Yaskawa INFORM job: clamp_07_08_23_cylinder_program.JBI

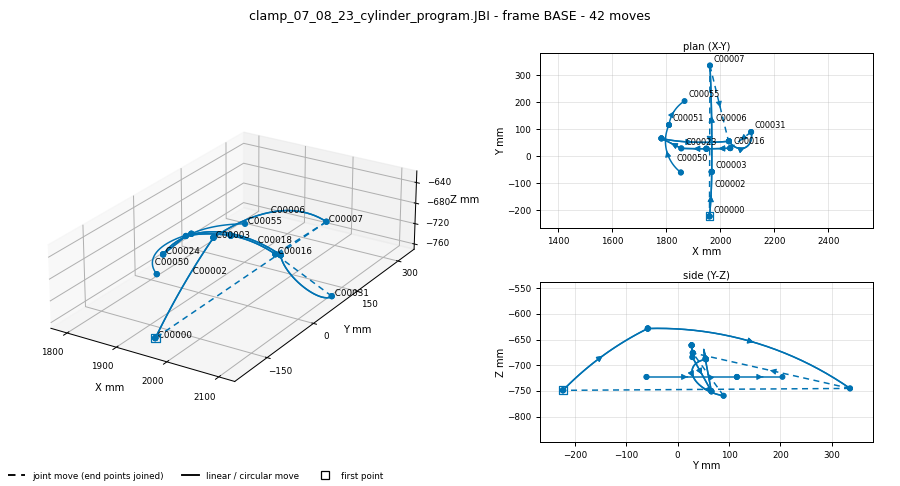
[picture p0: tool path of clamp_07_08_23_cylinder_program.JBI in frame BASE, 42 of 62 moves have a stored position in this frame; points joined in program order, loops and branches not executed]
/JOB
//NAME clamp_07_08_23_cylinder_program
//POS
///NPOS 56,0,56,0,0,0
///TOOL 0
///POSTYPE BASE
///RECTAN
///RCONF 0,0,0,0,0,0,0,0,0,0,0,0,0,0,0,0,0,0,0,0,0,0,0,0
C00000=1960.075828,-223.019615,-748.824454,180.000000,-60.000000,90.001386
C00001=1960.075828,-223.019615,-748.824454,180.000000,-60.000000,90.001386
C00002=1966.557197,-127.835510,-669.176522,-175.000000,-39.379629,92.626092
C00003=1968.376913,-58.034649,-628.612835,-161.404282,5.000000,5.000000
C00004=1968.376913,-58.034649,-628.612835,-161.404282,5.000000,5.000000
C00005=1968.376913,-58.034649,-628.612835,-161.404282,5.000000,5.000000
C00006=1968.142396,117.168535,-647.002737,151.969726,5.000000,-5.000000
C00007=1961.735097,335.262586,-745.090179,180.000000,-60.000000,-90.296572
C00008=1960.075828,-223.019615,-748.824454,180.000000,-60.000000,90.001386
C00009=1960.075828,-223.019615,-748.824454,180.000000,-60.000000,90.001386
C00010=1966.557197,-127.835510,-669.176522,-175.000000,-39.379629,92.626092
C00011=1968.376913,-58.034649,-628.612835,-161.404282,5.000000,5.000000
C00012=1968.376913,-58.034649,-628.612835,-161.404282,5.000000,5.000000
C00013=1968.376913,-58.034649,-628.612835,-161.404282,5.000000,5.000000
C00014=1968.142396,117.168535,-647.002737,151.969726,5.000000,-5.000000
C00015=1961.735097,335.262586,-745.090179,180.000000,-60.000000,-90.296572
C00016=2036.786677,29.436047,-676.031527,-174.048611,23.855296,5.000000
C00017=2036.786677,29.436047,-676.031527,-174.048611,23.855296,5.000000
C00018=1997.954834,27.911156,-664.054338,-174.328079,11.246992,5.000000
C00019=1948.764188,27.199700,-661.190386,-174.288511,-5.000000,-5.000000
C00020=1948.764188,27.199700,-661.190386,-174.288511,-5.000000,-5.000000
C00021=1948.764188,27.199700,-661.190386,-174.288511,-5.000000,-5.000000
C00022=1902.713206,27.551328,-668.774485,-173.853319,-18.487941,-5.000000
C00023=1855.573167,28.672798,-684.219428,175.000000,-33.996707,8.950518
C00024=1782.149442,65.644826,-750.764678,-180.000000,-60.000000,1.268123
C00025=1782.149442,65.644826,-750.764678,-180.000000,-60.000000,1.268123
C00026=1867.617170,53.257139,-684.581782,175.000000,-31.333075,9.869447
C00027=2031.930642,55.063888,-688.401258,-174.027335,24.456893,5.000000
C00028=2031.930642,55.063888,-688.401258,-174.027335,24.456893,5.000000
C00029=2031.930642,55.063888,-688.401258,-174.027335,24.456893,5.000000
C00030=2114.529672,61.982565,-750.948407,-175.000000,-59.425940,175.000000
C00031=2114.214530,89.330125,-759.380789,180.000000,-60.000000,-172.637609
C00032=2036.786677,29.436047,-676.031527,-174.048611,23.855296,5.000000
C00033=2036.786677,29.436047,-676.031527,-174.048611,23.855296,5.000000
C00034=1997.954834,27.911156,-664.054338,-174.328079,11.246992,5.000000
C00035=1948.764188,27.199700,-661.190386,-174.288511,-5.000000,-5.000000
C00036=1948.764188,27.199700,-661.190386,-174.288511,-5.000000,-5.000000
C00037=1948.764188,27.199700,-661.190386,-174.288511,-5.000000,-5.000000
C00038=1902.713206,27.551328,-668.774485,-173.853319,-18.487941,-5.000000
C00039=1855.573167,28.672798,-684.219428,175.000000,-33.996707,8.950518
C00040=1782.149442,65.644826,-750.764678,-180.000000,-60.000000,1.268123
C00041=1782.149442,65.644826,-750.764678,-180.000000,-60.000000,1.268123
C00042=1867.617170,53.257139,-684.581782,175.000000,-31.333075,9.869447
C00043=2031.930642,55.063888,-688.401258,-174.027335,24.456893,5.000000
C00044=2031.930642,55.063888,-688.401258,-174.027335,24.456893,5.000000
C00045=2031.930642,55.063888,-688.401258,-174.027335,24.456893,5.000000
C00046=2114.529672,61.982565,-750.948407,-175.000000,-59.425940,175.000000
C00047=2114.214530,89.330125,-759.380789,180.000000,-60.000000,-172.637609
C00048=1854.100788,-60.572273,-722.697460,180.000000,-60.000000,39.056159
C00049=1854.100788,-60.572273,-722.697460,180.000000,-60.000000,39.056159
C00050=1825.406210,-31.437250,-722.697460,180.000000,-60.000000,27.527976
C00051=1810.062104,115.232922,-722.697460,180.000000,-60.000000,-15.007935
C00052=1810.062104,115.232922,-722.697460,180.000000,-60.000000,-15.007935
C00053=1810.062104,115.232922,-722.697460,180.000000,-60.000000,-15.007935
C00054=1835.839436,175.302882,-722.697460,-180.000000,-60.000000,-33.491908
C00055=1867.753817,203.827510,-722.697460,180.000000,-60.000000,-45.587231
///POSTYPE PULSE
///PULSE
EX00000=0
EX00001=92160
EX00002=184320
EX00003=276480
///POSTYPE PULSE
///PULSE
EC00000=0
EC00001=0
EC00002=0
EC00003=0
EC00004=0
EC00005=0
EC00006=0
EC00007=0
EC00008=0
EC00009=0
EC00010=0
EC00011=0
EC00012=0
EC00013=0
EC00014=0
EC00015=0
EC00016=0
EC00017=0
EC00018=0
EC00019=0
EC00020=0
EC00021=0
EC00022=0
EC00023=0
EC00024=0
EC00025=0
EC00026=0
EC00027=0
EC00028=0
EC00029=0
EC00030=0
EC00031=0
EC00032=0
EC00033=0
EC00034=0
EC00035=0
EC00036=0
EC00037=0
EC00038=0
EC00039=0
EC00040=0
EC00041=0
EC00042=0
EC00043=0
EC00044=0
EC00045=0
EC00046=0
EC00047=0
EC00048=276480
EC00049=276480
EC00050=276480
EC00051=276480
EC00052=276480
EC00053=276480
EC00054=276480
EC00055=276480
//INST
///DATE 2023/08/07 12:02
///ATTR SC,RW,RJ
////FRAME BASE
///GROUP1 RB1,ST1
NOP
MOVJ P009 EX000 VJ=15.00
MOVJ C00000 EC00000 VJ=15.0
CALL JOB:SPYON
MOVC C00001 EC00001 V=150.0
MOVC C00002 EC00002 V=150.0
MOVC C00003 EC00003 V=150.0
MOVL C00004 EC00004 V=150.0
MOVC C00005 EC00005 V=150.0
MOVC C00006 EC00006 V=150.0
MOVC C00007 EC00007 V=150.0
CALL JOB:SPYOF
MOVJ C00008 EC00008 VJ=15.0
CALL JOB:SPYON
MOVC C00009 EC00009 V=150.0
MOVC C00010 EC00010 V=150.0
MOVC C00011 EC00011 V=150.0
MOVL C00012 EC00012 V=150.0
MOVC C00013 EC00013 V=150.0
MOVC C00014 EC00014 V=150.0
MOVC C00015 EC00015 V=150.0
CALL JOB:SPYOF
MOVJ C00016 EC00016 VJ=15.0
CALL JOB:SPYON
MOVC C00017 EC00017 V=150.0
MOVC C00018 EC00018 V=150.0
MOVC C00019 EC00019 V=150.0
MOVL C00020 EC00020 V=150.0
MOVC C00021 EC00021 V=150.0
MOVC C00022 EC00022 V=150.0
MOVC C00023 EC00023 V=150.0
MOVL C00024 EC00024 V=150.0
MOVC C00025 EC00025 V=150.0
MOVC C00026 EC00026 V=150.0
MOVC C00027 EC00027 V=150.0
MOVL C00028 EC00028 V=150.0
MOVC C00029 EC00029 V=150.0
MOVC C00030 EC00030 V=150.0
MOVC C00031 EC00031 V=150.0
CALL JOB:SPYOF
MOVJ C00032 EC00032 VJ=15.0
CALL JOB:SPYON
MOVC C00033 EC00033 V=150.0
MOVC C00034 EC00034 V=150.0
MOVC C00035 EC00035 V=150.0
MOVL C00036 EC00036 V=150.0
MOVC C00037 EC00037 V=150.0
MOVC C00038 EC00038 V=150.0
MOVC C00039 EC00039 V=150.0
MOVL C00040 EC00040 V=150.0
MOVC C00041 EC00041 V=150.0
MOVC C00042 EC00042 V=150.0
MOVC C00043 EC00043 V=150.0
MOVL C00044 EC00044 V=150.0
MOVC C00045 EC00045 V=150.0
MOVC C00046 EC00046 V=150.0
MOVC C00047 EC00047 V=150.0
CALL JOB:SPYOF
MOVJ P009 VJ=15.00
MOVJ P009 VJ=15.00
MOVJ P009 VJ=15.00
MOVJ P009 VJ=15.00
MOVJ C00048 EC00048 VJ=15.0
CALL JOB:SPYON
MOVC C00049 EC00049 V=150.0
MOVC C00050 EC00050 V=150.0
MOVC C00051 EC00051 V=150.0
MOVL C00052 EC00052 V=150.0
MOVC C00053 EC00053 V=150.0
MOVC C00054 EC00054 V=150.0
MOVC C00055 EC00055 V=150.0
CALL JOB:SPYOF
MOVJ P009 VJ=15.00
END
